// TIA Portal V19 export
FUNCTION "STOP CIP" : Void   // FC48, STL
TITLE = CIP ASEPTIC TANK
{ S7_Optimized_Access := 'TRUE' }
NAME : CIPTANK
VERSION : 0.0
// ****** REVISION HISTORY :
// 
// VERSION DATE         BY    DESCRIPTION
// --------------------------------------------------------------------------
// 00.00   4/2 1997   OPA   ORIGINAL FUNCTION BLOCK
//       
// THIS FUNCTION BLOCK IS USED FOR STOP CIP ON THE ASEPTIC TANK.
// 
// SOFTWARE SIMULATED IN OFFICE *******DATE*********
// stored: AutoNumber false
BEGIN

NETWORK
TITLE = CIP ASEPTIC TANK
// This network will stop all active functions and start drain of tank with 
// possible detergents.
      AN    "S0 STOP CIP TANK";
      R     "S1 STOP CIP TANK";
      R     "S2 STOP CIP TANK";
      R     "S3 STOP CIP TANK";
      R     "S4 STOP CIP TANK";
      BEC;
      A     "S1 STOP CIP TANK";
      JC    M001;
      R     "S.T.01.REQUEST LYE";  // STOP DOSING LYE IF ACTIVE
      R     "S.T.01.REQUEST ACID";  // STOP DOSING ACID IF ACTIVE
      R     "TANK CLEAN";
      R     "MY0158";
      R     "AutoTT0172/IP0157";
      R     "ManTT0172/IP0157";
      S     "MY0114";
      R     "CONTROL CIP TANK";
      S     "S1 STOP CIP TANK";
//;
      R     "MY0904";
      R     "MY0907";
      R     "MY0912";
//;
      BEU;
M001: NOP   0;

NETWORK
TITLE = WAIT FOR DRAIN TANK
// When the CIP tank has been drained, then start controlling water level in
// CIP-tank again.
      A     "S2 STOP CIP TANK";
      JC    c017;
      AN    "MM0139";
      S     "TIM34";
      S     "S2 STOP CIP TANK";
      S     "S3 STOP CIP TANK";
      R     "AutoPT0167/IP0149";
      R     "ManPT0167/IP0149";
      BEC;
      A     "B01.42";
      BEC;
      S     "CONTROL CIP TANK";
      S     "TIM33";
      S     "S2 STOP CIP TANK";
      BEU;
c017: NOP   0;

NETWORK
TITLE = FINAL RINSE/FLUSH OUT DETERGENTS
// Wait for water flush timer, then stop pumps and reset
      A     "S3 STOP CIP TANK";
      JC    c018;
      A     "T 33 WATER 3";
      BEC;
      R     "CONTROL CIP TANK";
      R     "MM0139";
      R     "MY0103";
      R     "MY0104";
      R     "AutoPT0167/IP0149";
      R     "ManPT0167/IP0149";
      S     "TIM34";
      S     "PULSE 01.13 CIP";
      S     "S3 STOP CIP TANK";
      BEU;
c018: NOP   0;

NETWORK
TITLE = BLOW OUT
// Comment
      A     "S4 STOP CIP TANK";
      JC    c019;
      A     "T 34 BLOW OUT CIP";
      BEC;
      R     "S0 STOP CIP TANK";
      BEU;
c019: NOP   0;
END_FUNCTION
